% RSLogix 500 project HEATER DIGITAL INPUTS.RSS, saved by version 8.30.00.16 %
PROJECT "UNTITLED"    % processor: Bul.1763 MicroLogix 1100 Series B %

PROGRAM FILES
  LAD 2 "MAIN"  3 rungs
  LAD 3 "IO"  3 rungs  % IO %
  LAD 4 "CONTROL"  7 rungs

DATA FILES
  O0 OUTPUT  9 elements
  I1 INPUT  16 elements
  S2 STATUS  66 elements
  B3 BINARY  1 elements
  T4 TIMER  1 elements
  C5 COUNTER  1 elements
  R6 CONTROL  1 elements
  N7 INTEGER  1 elements
  F8 FLOAT  1 elements

LADDER 2 "MAIN"
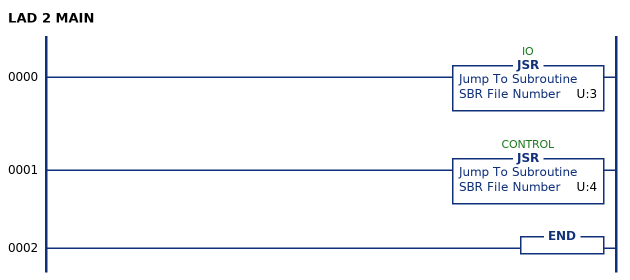
% Rung: 0 %  % edit flag set %
SOR JSR U:3 EOR
%   U:3  "IO" %
% Rung: 1 %  % edit flag set %
SOR JSR U:4 EOR
%   U:4  "CONTROL" %
% Rung: 2 %
SOR END EOR

LADDER 3 "IO"    % IO %
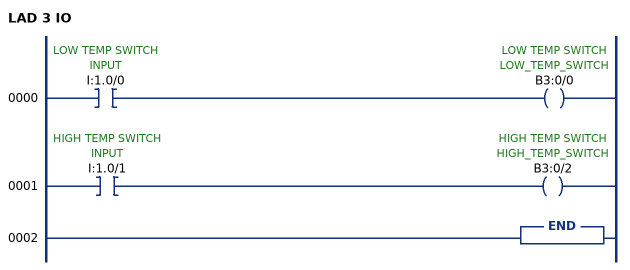
% Rung: 0 %  % edit flag set %
SOR XIC I:1.0/0 OTE B3:0/0 EOR
%   I:1.0/0  "LOW TEMP SWITCH INPUT" %
%   B3:0/0  LOW_TEMP_SWITCH  "LOW TEMP SWITCH" %
% Rung: 1 %  % edit flag set %
SOR XIC I:1.0/1 OTE B3:0/2 EOR
%   I:1.0/1  "HIGH TEMP SWITCH INPUT" %
%   B3:0/2  HIGH_TEMP_SWITCH  "HIGH TEMP SWITCH" %
% Rung: 2 %
SOR END EOR

LADDER 4 "CONTROL"
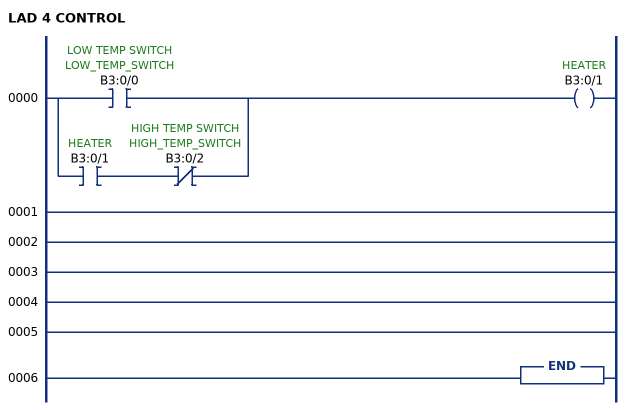
% Rung: 0 %  % edit flag set %
SOR BST XIC B3:0/0 NXB XIC B3:0/1 XIO B3:0/2 BND OTE B3:0/1 EOR
%   B3:0/0  LOW_TEMP_SWITCH  "LOW TEMP SWITCH" %
%   B3:0/1  "HEATER" %
%   B3:0/2  HIGH_TEMP_SWITCH  "HIGH TEMP SWITCH" %
% Rung: 1 %  % edit flag set %
SOR EOR
% Rung: 2 %  % edit flag set %
SOR EOR
% Rung: 3 %  % edit flag set %
SOR EOR
% Rung: 4 %  % edit flag set %
SOR EOR
% Rung: 5 %  % edit flag set %
SOR EOR
% Rung: 6 %
SOR END EOR

OTHER DOCUMENTED ADDRESSES
  I:0.0/0  "LOW TEMP SWITCH INPUT"
  I:0.0/1  "HIGH TEM SWITCH INPUT"
  O:2.0/0  "HEATER OUTPUT"
